{attribute 'qualified_only'}
{attribute 'strict'}
TYPE eIcon :
(
	Emg			:= 0,
	DoorOpen	:= 1,
	AirOk		:= 2,
	HydraulicOk	:= 3,
	EquipmentOk	:= 4,
	Home		:= 5,
	Connection	:= 6,
	End			:= 16
);
END_TYPE

(* stored: Version 1.1.0.1, ProductVersion 3.1.4024.13
   EnumerationTextList eIcon: Id {1f95683c-b48b-4382-b0f2-7d414508d639} *)
